(* PLC project interlocking_NUC1.project, CODESYS CODESYS V3.5 SP21 Patch 1 *)
(* stored: creationDateTime 2025-07-24T17:00:33.8424402, modificationDateTime 2025-07-24T17:00:18.702934 *)

PROGRAM PLC_PRG
  VAR_INPUT
    Input1 : BOOL := FALSE;  (* AA1D1Q01Q1QA1/CSWI1.Pos *)
    Input2 : BOOL := FALSE;  (* AA1D1Q01Q1QB2/CSWI1.Pos *)
    Input3 : BOOL := FALSE;  (* AA1D1Q05Q1CBSW/XCBR1.Pos.stVal *)
    Input4 : BOOL := FALSE;  (* AA1D1Q05Q1CBSW/XSWI1.Pos.stVal *)
    Input5 : BOOL := FALSE;  (* AA1D1Q05Q1CBSW/XSWI2.Pos.stVal *)
    Input6 : BOOL := FALSE;  (* AA1D1Q05Q1CBSW/XSWI3.Pos.stVal *)
  END_VAR
  VAR_OUTPUT
    Output1 : BOOL := FALSE;  (* AA1D1Q01Q1QB1/CILO1.EnaCls *)
  END_VAR

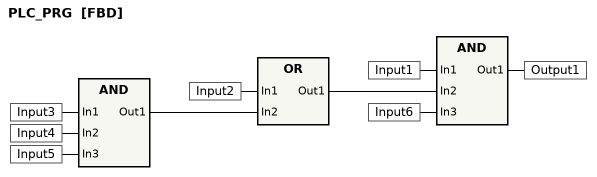
(* FBD diagram, written out as Structured Text *)
Output1 := Input1 AND (Input2 OR Input3 AND Input4 AND Input5) AND Input6;
END_PROGRAM
